LIN {X 0,Y 180.514,Z 1092.741,A -85,B 0,C 180,E1 5202.314,E2 5202.314} C_VEL
LIN {X 0,Y 161.576,Z 1104.142,A -85,B 0,C 180,E1 5198.165,E2 5198.165} C_VEL
LIN {X 0,Y 144.452,Z 1113.156,A -85,B 0,C 180,E1 5193.245,E2 5193.245} C_VEL
LIN {X 0,Y 126.484,Z 1121.616,A -85,B 0,C 180,E1 5186.105,E2 5186.105} C_VEL
LIN {X 0,Y 112.708,Z 1127.399,A -85,B 0,C 180,E1 5178.177,E2 5178.177} C_VEL
LIN {X 0,Y 100.075,Z 1132.394,A -85,B 0,C 180,E1 5166.833,E2 5166.833} C_VEL
LIN {X 0,Y 92.274,Z 1135.383,A -85,B 0,C 180,E1 5154.316,E2 5154.316} C_VEL
LIN {X 0,Y 88.588,Z 1137.104,A -85,B 0,C 180,E1 5140.404,E2 5140.404} C_VEL
LIN {X 0,Y 88.071,Z 1137.45,A -85,B 0,C 180,E1 5129.349,E2 5129.349} C_VEL
LIN {X 0,Y 88.847,Z 1136.939,A -85,B 0,C 180,E1 5117.653,E2 5117.653} C_VEL
LIN {X 0,Y 92.778,Z 1135.217,A -85,B 0,C 180,E1 5104.463,E2 5104.463} C_VEL
LIN {X 0,Y 101.858,Z 1131.792,A -85,B 0,C 180,E1 5091.078,E2 5091.078} C_VEL
LIN {X 0,Y 114.473,Z 1126.766,A -85,B 0,C 180,E1 5080.542,E2 5080.542} C_VEL
LIN {X 0,Y 130.71,Z 1119.847,A -85,B 0,C 180,E1 5071.884,E2 5071.884} C_VEL
LIN {X 0,Y 146.756,Z 1112.133,A -85,B 0,C 180,E1 5065.926,E2 5065.926} C_VEL
LIN {X 0,Y 165.729,Z 1101.922,A -85,B 0,C 180,E1 5060.745,E2 5060.745} C_VEL
LIN {X 0,Y 183.093,Z 1091.275,A -85,B 0,C 180,E1 5057.119,E2 5057.119} C_VEL
LIN {X 0,Y 202.882,Z 1077.554,A -85,B 0,C 180,E1 5053.854,E2 5053.854} C_VEL
LIN {X 0,Y 219.478,Z 1064.484,A -85,B 0,C 180,E1 5051.623,E2 5051.623} C_VEL
LIN {X 0,Y 238.252,Z 1047.708,A -85,B 0,C 180,E1 5049.514,E2 5049.514} C_VEL
LIN {X 0,Y 253.475,Z 1032.291,A -85,B 0,C 180,E1 5048.055,E2 5048.055} C_VEL
LIN {X 0,Y 269.807,Z 1013.44,A -85,B 0,C 180,E1 5046.686,E2 5046.686} C_VEL
LIN {X 0,Y 282.88,Z 996.295,A -85,B 0,C 180,E1 5045.721,E2 5045.721} C_VEL
LIN {X 0,Y 296.514,Z 975.768,A -85,B 0,C 180,E1 5044.812,E2 5044.812} C_VEL
LIN {X 0,Y 307.276,Z 957.078,A -85,B 0,C 180,E1 5044.155,E2 5044.155} C_VEL
LIN {X 0,Y 318.569,Z 934.064,A -85,B 0,C 180,E1 5043.522,E2 5043.522} C_VEL
LIN {X 0,Y 326.941,Z 913.681,A -85,B 0,C 180,E1 5043.088,E2 5043.088} C_VEL
LIN {X 0,Y 335.084,Z 889.205,A -85,B 0,C 180,E1 5042.688,E2 5042.688} C_VEL
LIN {X 0,Y 340.736,Z 867.45,A -85,B 0,C 180,E1 5042.416,E2 5042.416} C_VEL
LIN {X 0,Y 345.393,Z 842.416,A -85,B 0,C 180,E1 5042.144,E2 5042.144} C_VEL
LIN {X 0,Y 352.177,Z 788.71,A -85,B 0,C 180,E1 5041.569,E2 5041.569} C_VEL
LIN {X 0,Y 344.618,Z 847.74,A -85,B 0,C 180,E1 5040.925,E2 5040.925} C_VEL
LIN {X 0,Y 339.705,Z 871.733,A -85,B 0,C 180,E1 5040.649,E2 5040.649} C_VEL
LIN {X 0,Y 333.471,Z 894.758,A -85,B 0,C 180,E1 5040.334,E2 5040.334} C_VEL
LIN {X 0,Y 325.466,Z 917.45,A -85,B 0,C 180,E1 5039.929,E2 5039.929} C_VEL
LIN {X 0,Y 315.983,Z 939.81,A -85,B 0,C 180,E1 5039.422,E2 5039.422} C_VEL
LIN {X 0,Y 305.532,Z 960.244,A -85,B 0,C 180,E1 5038.827,E2 5038.827} C_VEL
LIN {X 0,Y 293.092,Z 981.341,A -85,B 0,C 180,E1 5038.045,E2 5038.045} C_VEL
LIN {X 0,Y 279.658,Z 1000.791,A -85,B 0,C 180,E1 5037.131,E2 5037.131} C_VEL
LIN {X 0,Y 264.625,Z 1019.965,A -85,B 0,C 180,E1 5035.975,E2 5035.975} C_VEL
LIN {X 0,Y 249.554,Z 1036.734,A -85,B 0,C 180,E1 5034.669,E2 5034.669} C_VEL
LIN {X 0,Y 232.717,Z 1053.447,A -85,B 0,C 180,E1 5032.987,E2 5032.987} C_VEL
LIN {X 0,Y 215.64,Z 1068.312,A -85,B 0,C 180,E1 5030.988,E2 5030.988} C_VEL
LIN {X 0,Y 210.299,Z 1072.727,A -85,B 0,C 180,E1 5030.284,E2 5030.284} C_VEL
LIN {X 0,Y 204.27,Z 1077.246,A -85,B 0,C 180,E1 5029.757,E2 5029.757} C_VEL
LIN {X 0,Y 187.534,Z 1088.286,A -85,B 0,C 180,E1 5029.208,E2 5029.208} C_VEL
LIN {X 0,Y 181.234,Z 1092.239,A -85,B 0,C 180,E1 5028.527,E2 5028.527} C_VEL
LIN {X 0,Y 163.079,Z 1103.329,A -85,B 0,C 180,E1 5025.077,E2 5025.077} C_VEL
LIN {X 0,Y 142.378,Z 1114.455,A -85,B 0,C 180,E1 5019.872,E2 5019.872} C_VEL
LIN {X 0,Y 125.566,Z 1122.468,A -85,B 0,C 180,E1 5014.025,E2 5014.025} C_VEL
LIN {X 0,Y 108.268,Z 1129.827,A -85,B 0,C 180,E1 5005.28,E2 5005.28} C_VEL
LIN {X 0,Y 95.103,Z 1135.026,A -85,B 0,C 180,E1 4994.783,E2 4994.783} C_VEL
LIN {X 0,Y 84.698,Z 1139.105,A -85,B 0,C 180,E1 4979.724,E2 4979.724} C_VEL
LIN {X 0,Y 80.754,Z 1140.969,A -85,B 0,C 180,E1 4966.546,E2 4966.546} C_VEL
LIN {X 0,Y 79.997,Z 1141.711,A -85,B 0,C 180,E1 4955.019,E2 4955.019} C_VEL
LIN {X 0,Y 80.026,Z 1141.802,A -85,B 0,C 180,E1 4947.852,E2 4947.852} C_VEL
LIN {X 0,Y 80.375,Z 1141.239,A -85,B 0,C 180,E1 4936.328,E2 4936.328} C_VEL
LIN {X 0,Y 83.833,Z 1139.429,A -85,B 0,C 180,E1 4922.279,E2 4922.279} C_VEL
LIN {X 0,Y 92.595,Z 1135.983,A -85,B 0,C 180,E1 4907.97,E2 4907.97} C_VEL
LIN {X 0,Y 105.649,Z 1130.794,A -85,B 0,C 180,E1 4896.441,E2 4896.441} C_VEL
LIN {X 0,Y 121.066,Z 1124.38,A -85,B 0,C 180,E1 4887.905,E2 4887.905} C_VEL
LIN {X 0,Y 139.45,Z 1115.772,A -85,B 0,C 180,E1 4881.009,E2 4881.009} C_VEL
LIN {X 0,Y 158.123,Z 1106.034,A -85,B 0,C 180,E1 4876.018,E2 4876.018} C_VEL
LIN {X 0,Y 176.98,Z 1094.75,A -85,B 0,C 180,E1 4872.201,E2 4872.201} C_VEL
LIN {X 0,Y 195.527,Z 1082.343,A -85,B 0,C 180,E1 4869.258,E2 4869.258} C_VEL
LIN {X 0,Y 214.497,Z 1067.805,A -85,B 0,C 180,E1 4866.823,E2 4866.823} C_VEL
LIN {X 0,Y 232.288,Z 1052.516,A -85,B 0,C 180,E1 4864.939,E2 4864.939} C_VEL
LIN {X 0,Y 249.412,Z 1035.598,A -85,B 0,C 180,E1 4863.395,E2 4863.395} C_VEL
LIN {X 0,Y 265.655,Z 1017.529,A -85,B 0,C 180,E1 4862.13,E2 4862.13} C_VEL
LIN {X 0,Y 280.026,Z 999.098,A -85,B 0,C 180,E1 4861.142,E2 4861.142} C_VEL
LIN {X 0,Y 293.973,Z 978.764,A -85,B 0,C 180,E1 4860.288,E2 4860.288} C_VEL
LIN {X 0,Y 305.646,Z 958.886,A -85,B 0,C 180,E1 4859.625,E2 4859.625} C_VEL
LIN {X 0,Y 316.509,Z 937.477,A -85,B 0,C 180,E1 4859.065,E2 4859.065} C_VEL
LIN {X 0,Y 325.559,Z 915.956,A -85,B 0,C 180,E1 4858.631,E2 4858.631} C_VEL
LIN {X 0,Y 330.238,Z 903.054,A -85,B 0,C 180,E1 4858.407,E2 4858.407} C_VEL
LIN {X 0,Y 321.662,Z 925.806,A -85,B 0,C 180,E1 4858.004,E2 4858.004} C_VEL
LIN {X 0,Y 311.963,Z 946.817,A -85,B 0,C 180,E1 4857.526,E2 4857.526} C_VEL
LIN {X 0,Y 300.406,Z 968.233,A -85,B 0,C 180,E1 4856.909,E2 4856.909} C_VEL
LIN {X 0,Y 288.154,Z 987.533,A -85,B 0,C 180,E1 4856.2,E2 4856.2} C_VEL
LIN {X 0,Y 273.899,Z 1007.211,A -85,B 0,C 180,E1 4855.283,E2 4855.283} C_VEL
LIN {X 0,Y 259.287,Z 1024.684,A -85,B 0,C 180,E1 4854.229,E2 4854.229} C_VEL
LIN {X 0,Y 242.854,Z 1042.089,A -85,B 0,C 180,E1 4852.868,E2 4852.868} C_VEL
LIN {X 0,Y 226.575,Z 1057.152,A -85,B 0,C 180,E1 4851.314,E2 4851.314} C_VEL
LIN {X 0,Y 208.615,Z 1071.963,A -85,B 0,C 180,E1 4849.286,E2 4849.286} C_VEL
LIN {X 0,Y 190.964,Z 1084.666,A -85,B 0,C 180,E1 4846.882,E2 4846.882} C_VEL
LIN {X 0,Y 171.93,Z 1096.865,A -85,B 0,C 180,E1 4843.657,E2 4843.657} C_VEL
LIN {X 0,Y 153.55,Z 1107.072,A -85,B 0,C 180,E1 4839.67,E2 4839.67} C_VEL
LIN {X 0,Y 134.485,Z 1116.453,A -85,B 0,C 180,E1 4834.11,E2 4834.11} C_VEL
LIN {X 0,Y 117.722,Z 1123.611,A -85,B 0,C 180,E1 4827.233,E2 4827.233} C_VEL
LIN {X 0,Y 101.608,Z 1129.793,A -85,B 0,C 180,E1 4817.233,E2 4817.233} C_VEL
LIN {X 0,Y 90.459,Z 1133.686,A -85,B 0,C 180,E1 4805.862,E2 4805.862} C_VEL
LIN {X 0,Y 82.662,Z 1136.478,A -85,B 0,C 180,E1 4790.536,E2 4790.536} C_VEL
LIN {X 0,Y 80.264,Z 1137.458,A -85,B 0,C 180,E1 4777.156,E2 4777.156} C_VEL
LIN {X 0,Y 80.087,Z 1137.594,A -85,B 0,C 180,E1 4767.137,E2 4767.137} C_VEL
LIN {X 0,Y 81.399,Z 1136.957,A -85,B 0,C 180,E1 4754.321,E2 4754.321} C_VEL
LIN {X 0,Y 86.185,Z 1135.212,A -85,B 0,C 180,E1 4740.839,E2 4740.839} C_VEL
LIN {X 0,Y 97.246,Z 1131.404,A -85,B 0,C 180,E1 4726.457,E2 4726.457} C_VEL
LIN {X 0,Y 110.682,Z 1126.484,A -85,B 0,C 180,E1 4716.484,E2 4716.484} C_VEL
LIN {X 0,Y 128.899,Z 1119.024,A -85,B 0,C 180,E1 4707.832,E2 4707.832} C_VEL
LIN {X 0,Y 145.872,Z 1111.156,A -85,B 0,C 180,E1 4702.275,E2 4702.275} C_VEL
LIN {X 0,Y 165.655,Z 1100.621,A -85,B 0,C 180,E1 4697.505,E2 4697.505} C_VEL
LIN {X 0,Y 183.74,Z 1089.709,A -85,B 0,C 180,E1 4694.175,E2 4694.175} C_VEL
LIN {X 0,Y 202.953,Z 1076.4,A -85,B 0,C 180,E1 4691.357,E2 4691.357} C_VEL
LIN {X 0,Y 220.831,Z 1062.434,A -85,B 0,C 180,E1 4689.221,E2 4689.221} C_VEL
LIN {X 0,Y 238.175,Z 1046.883,A -85,B 0,C 180,E1 4687.478,E2 4687.478} C_VEL
LIN {X 0,Y 254.406,Z 1030.543,A -85,B 0,C 180,E1 4686.084,E2 4686.084} C_VEL
LIN {X 0,Y 269.963,Z 1012.521,A -85,B 0,C 180,E1 4684.912,E2 4684.912} C_VEL
LIN {X 0,Y 284.154,Z 993.949,A -85,B 0,C 180,E1 4683.976,E2 4683.976} C_VEL
LIN {X 0,Y 297.427,Z 973.701,A -85,B 0,C 180,E1 4683.18,E2 4683.18} C_VEL
LIN {X 0,Y 309.271,Z 952.974,A -85,B 0,C 180,E1 4682.537,E2 4682.537} C_VEL
LIN {X 0,Y 319.664,Z 931.164,A -85,B 0,C 180,E1 4682.012,E2 4682.012} C_VEL
LIN {X 0,Y 328.842,Z 908.282,A -85,B 0,C 180,E1 4681.586,E2 4681.586} C_VEL
LIN {X 0,Y 329.621,Z 905.974,A -85,B 0,C 180,E1 4681.548,E2 4681.548} C_VEL
LIN {X 0,Y 320.528,Z 929.195,A -85,B 0,C 180,E1 4681.122,E2 4681.122} C_VEL
LIN {X 0,Y 311.488,Z 948.495,A -85,B 0,C 180,E1 4680.664,E2 4680.664} C_VEL
LIN {X 0,Y 298.969,Z 971.183,A -85,B 0,C 180,E1 4679.988,E2 4679.988} C_VEL
LIN {X 0,Y 286.993,Z 989.827,A -85,B 0,C 180,E1 4679.284,E2 4679.284} C_VEL
LIN {X 0,Y 271.594,Z 1010.601,A -85,B 0,C 180,E1 4678.286,E2 4678.286} C_VEL
LIN {X 0,Y 256.782,Z 1028.09,A -85,B 0,C 180,E1 4677.189,E2 4677.189} C_VEL
LIN {X 0,Y 239.636,Z 1045.793,A -85,B 0,C 180,E1 4675.745,E2 4675.745} C_VEL
LIN {X 0,Y 222.674,Z 1061.316,A -85,B 0,C 180,E1 4674.072,E2 4674.072} C_VEL
LIN {X 0,Y 204.021,Z 1076.268,A -85,B 0,C 180,E1 4671.887,E2 4671.887} C_VEL
LIN {X 0,Y 185.27,Z 1089.642,A -85,B 0,C 180,E1 4669.187,E2 4669.187} C_VEL
LIN {X 0,Y 181.234,Z 1092.239,A -85,B 0,C 180,E1 4668.527,E2 4668.527} C_VEL
LIN {X 0,Y 174.874,Z 1096.127,A -85,B 0,C 180,E1 4667.781,E2 4667.781} C_VEL
LIN {X 0,Y 156.317,Z 1105.93,A -85,B 0,C 180,E1 4666.648,E2 4666.648} C_VEL
LIN {X 0,Y 150.773,Z 1108.689,A -85,B 0,C 180,E1 4665.773,E2 4665.773} C_VEL
LIN {X 0,Y 131.4,Z 1118.23,A -85,B 0,C 180,E1 4660.663,E2 4660.663} C_VEL
LIN {X 0,Y 112.711,Z 1126.128,A -85,B 0,C 180,E1 4653.637,E2 4653.637} C_VEL
LIN {X 0,Y 96.223,Z 1132.453,A -85,B 0,C 180,E1 4644.148,E2 4644.148} C_VEL
LIN {X 0,Y 83.081,Z 1136.987,A -85,B 0,C 180,E1 4631.447,E2 4631.447} C_VEL
LIN {X 0,Y 74.722,Z 1140.085,A -85,B 0,C 180,E1 4615.354,E2 4615.354} C_VEL
LIN {X 0,Y 72.037,Z 1141.397,A -85,B 0,C 180,E1 4598.783,E2 4598.783} C_VEL
LIN {X 0,Y 72.05,Z 1141.64,A -85,B 0,C 180,E1 4589.205,E2 4589.205} C_VEL
LIN {X 0,Y 72.206,Z 1141.284,A -85,B 0,C 180,E1 4578.011,E2 4578.011} C_VEL
LIN {X 0,Y 76.063,Z 1139.453,A -85,B 0,C 180,E1 4560.896,E2 4560.896} C_VEL
LIN {X 0,Y 84.556,Z 1136.434,A -85,B 0,C 180,E1 4546.696,E2 4546.696} C_VEL
LIN {X 0,Y 99.622,Z 1131.08,A -85,B 0,C 180,E1 4533.506,E2 4533.506} C_VEL
LIN {X 0,Y 115.63,Z 1124.862,A -85,B 0,C 180,E1 4525.07,E2 4525.07} C_VEL
LIN {X 0,Y 135.793,Z 1115.982,A -85,B 0,C 180,E1 4518.015,E2 4518.015} C_VEL
LIN {X 0,Y 154.225,Z 1106.745,A -85,B 0,C 180,E1 4513.467,E2 4513.467} C_VEL
LIN {X 0,Y 174.479,Z 1095.102,A -85,B 0,C 180,E1 4509.705,E2 4509.705} C_VEL
LIN {X 0,Y 192.455,Z 1083.398,A -85,B 0,C 180,E1 4507.097,E2 4507.097} C_VEL
LIN {X 0,Y 211.73,Z 1069.117,A -85,B 0,C 180,E1 4504.83,E2 4504.83} C_VEL
LIN {X 0,Y 229.316,Z 1054.363,A -85,B 0,C 180,E1 4503.122,E2 4503.122} C_VEL
LIN {X 0,Y 247.593,Z 1036.838,A -85,B 0,C 180,E1 4501.62,E2 4501.62} C_VEL
LIN {X 0,Y 262.984,Z 1020.126,A -85,B 0,C 180,E1 4500.529,E2 4500.529} C_VEL
LIN {X 0,Y 278.479,Z 1000.799,A -85,B 0,C 180,E1 4499.559,E2 4499.559} C_VEL
LIN {X 0,Y 291.731,Z 981.983,A -85,B 0,C 180,E1 4498.822,E2 4498.822} C_VEL
LIN {X 0,Y 299.524,Z 969.498,A -85,B 0,C 180,E1 4498.416,E2 4498.416} C_VEL
LIN {X 0,Y 287.188,Z 988.671,A -85,B 0,C 180,E1 4497.766,E2 4497.766} C_VEL
LIN {X 0,Y 271.876,Z 1009.318,A -85,B 0,C 180,E1 4496.875,E2 4496.875} C_VEL
LIN {X 0,Y 257.62,Z 1026.066,A -85,B 0,C 180,E1 4495.939,E2 4495.939} C_VEL
LIN {X 0,Y 240.036,Z 1044.183,A -85,B 0,C 180,E1 4494.612,E2 4494.612} C_VEL
LIN {X 0,Y 223.564,Z 1059.076,A -85,B 0,C 180,E1 4493.168,E2 4493.168} C_VEL
LIN {X 0,Y 204.401,Z 1074.28,A -85,B 0,C 180,E1 4491.17,E2 4491.17} C_VEL
LIN {X 0,Y 186.475,Z 1086.779,A -85,B 0,C 180,E1 4488.891,E2 4488.891} C_VEL
LIN {X 0,Y 166.165,Z 1099.122,A -85,B 0,C 180,E1 4485.654,E2 4485.654} C_VEL
LIN {X 0,Y 147.885,Z 1108.844,A -85,B 0,C 180,E1 4481.879,E2 4481.879} C_VEL
LIN {X 0,Y 127.81,Z 1118.057,A -85,B 0,C 180,E1 4476.252,E2 4476.252} C_VEL
LIN {X 0,Y 110.494,Z 1125.014,A -85,B 0,C 180,E1 4469.281,E2 4469.281} C_VEL
LIN {X 0,Y 93.986,Z 1130.73,A -85,B 0,C 180,E1 4459.056,E2 4459.056} C_VEL
LIN {X 0,Y 81.705,Z 1134.671,A -85,B 0,C 180,E1 4445.974,E2 4445.974} C_VEL
LIN {X 0,Y 74.127,Z 1136.983,A -85,B 0,C 180,E1 4429.226,E2 4429.226} C_VEL
LIN {X 0,Y 72.169,Z 1137.731,A -85,B 0,C 180,E1 4415.566,E2 4415.566} C_VEL
LIN {X 0,Y 72.11,Z 1137.783,A -85,B 0,C 180,E1 4406.024,E2 4406.024} C_VEL
LIN {X 0,Y 73.663,Z 1137.168,A -85,B 0,C 180,E1 4392.625,E2 4392.625} C_VEL
LIN {X 0,Y 79.198,Z 1135.424,A -85,B 0,C 180,E1 4377.977,E2 4377.977} C_VEL
LIN {X 0,Y 91.511,Z 1131.617,A -85,B 0,C 180,E1 4362.939,E2 4362.939} C_VEL
LIN {X 0,Y 105.313,Z 1126.945,A -85,B 0,C 180,E1 4353.33,E2 4353.33} C_VEL
LIN {X 0,Y 124.481,Z 1119.586,A -85,B 0,C 180,E1 4344.814,E2 4344.814} C_VEL
LIN {X 0,Y 142.11,Z 1111.77,A -85,B 0,C 180,E1 4339.467,E2 4339.467} C_VEL
LIN {X 0,Y 162.482,Z 1101.351,A -85,B 0,C 180,E1 4334.948,E2 4334.948} C_VEL
LIN {X 0,Y 180.834,Z 1090.59,A -85,B 0,C 180,E1 4331.848,E2 4331.848} C_VEL
LIN {X 0,Y 200.88,Z 1077.094,A -85,B 0,C 180,E1 4329.165,E2 4329.165} C_VEL
LIN {X 0,Y 217.753,Z 1064.194,A -85,B 0,C 180,E1 4327.322,E2 4327.322} C_VEL
LIN {X 0,Y 236.117,Z 1048.215,A -85,B 0,C 180,E1 4325.636,E2 4325.636} C_VEL
LIN {X 0,Y 251.719,Z 1032.814,A -85,B 0,C 180,E1 4324.411,E2 4324.411} C_VEL
LIN {X 0,Y 268.408,Z 1014.018,A -85,B 0,C 180,E1 4323.267,E2 4323.267} C_VEL
LIN {X 0,Y 281.731,Z 996.907,A -85,B 0,C 180,E1 4322.465,E2 4322.465} C_VEL
LIN {X 0,Y 296.097,Z 975.666,A -85,B 0,C 180,E1 4321.686,E2 4321.686} C_VEL
LIN {X 0,Y 298.821,Z 971.242,A -85,B 0,C 180,E1 4321.534,E2 4321.534} C_VEL
LIN {X 0,Y 286.504,Z 990.236,A -85,B 0,C 180,E1 4320.884,E2 4320.884} C_VEL
LIN {X 0,Y 271.292,Z 1010.529,A -85,B 0,C 180,E1 4320,E2 4320} C_VEL
LIN {X 0,Y 256.462,Z 1027.865,A -85,B 0,C 180,E1 4319.015,E2 4319.015} C_VEL
LIN {X 0,Y 239.166,Z 1045.537,A -85,B 0,C 180,E1 4317.708,E2 4317.708} C_VEL
LIN {X 0,Y 222.457,Z 1060.645,A -85,B 0,C 180,E1 4316.234,E2 4316.234} C_VEL
LIN {X 0,Y 203.02,Z 1076.033,A -85,B 0,C 180,E1 4314.194,E2 4314.194} C_VEL
LIN {X 0,Y 183.897,Z 1089.41,A -85,B 0,C 180,E1 4311.721,E2 4311.721} C_VEL
LIN {X 0,Y 164.267,Z 1101.321,A -85,B 0,C 180,E1 4308.524,E2 4308.524} C_VEL
LIN {X 0,Y 150.773,Z 1108.689,A -85,B 0,C 180,E1 4305.773,E2 4305.773} C_VEL
LIN {X 0,Y 144.235,Z 1111.943,A -85,B 0,C 180,E1 4304.698,E2 4304.698} C_VEL
LIN {X 0,Y 126.056,Z 1119.34,A -85,B 0,C 180,E1 4302.811,E2 4302.811} C_VEL
LIN {X 0,Y 119.505,Z 1121.914,A -85,B 0,C 180,E1 4301.308,E2 4301.308} C_VEL
LIN {X 0,Y 99.764,Z 1129.392,A -85,B 0,C 180,E1 4293.127,E2 4293.127} C_VEL
LIN {X 0,Y 84.188,Z 1134.592,A -85,B 0,C 180,E1 4282.727,E2 4282.727} C_VEL
LIN {X 0,Y 70.92,Z 1138.676,A -85,B 0,C 180,E1 4266.31,E2 4266.31} C_VEL
LIN {X 0,Y 65.157,Z 1140.616,A -85,B 0,C 180,E1 4249.731,E2 4249.731} C_VEL
LIN {X 0,Y 64.002,Z 1141.34,A -85,B 0,C 180,E1 4234.48,E2 4234.48} C_VEL
LIN {X 0,Y 64.01,Z 1141.358,A -85,B 0,C 180,E1 4226.418,E2 4226.418} C_VEL
LIN {X 0,Y 64.853,Z 1140.74,A -85,B 0,C 180,E1 4212.04,E2 4212.04} C_VEL
LIN {X 0,Y 70.129,Z 1138.878,A -85,B 0,C 180,E1 4195.227,E2 4195.227} C_VEL
LIN {X 0,Y 81.732,Z 1135.362,A -85,B 0,C 180,E1 4179.506,E2 4179.506} C_VEL
LIN {X 0,Y 97.477,Z 1130.095,A -85,B 0,C 180,E1 4168.095,E2 4168.095} C_VEL
LIN {X 0,Y 115.923,Z 1123.31,A -85,B 0,C 180,E1 4159.918,E2 4159.918} C_VEL
LIN {X 0,Y 136.017,Z 1114.58,A -85,B 0,C 180,E1 4153.983,E2 4153.983} C_VEL
LIN {X 0,Y 156.238,Z 1104.587,A -85,B 0,C 180,E1 4149.744,E2 4149.744} C_VEL
LIN {X 0,Y 176.147,Z 1093.122,A -85,B 0,C 180,E1 4146.595,E2 4146.595} C_VEL
LIN {X 0,Y 196.539,Z 1079.763,A -85,B 0,C 180,E1 4144.084,E2 4144.084} C_VEL
LIN {X 0,Y 214.154,Z 1066.531,A -85,B 0,C 180,E1 4142.323,E2 4142.323} C_VEL
LIN {X 0,Y 233.22,Z 1050.344,A -85,B 0,C 180,E1 4140.737,E2 4140.737} C_VEL
LIN {X 0,Y 249.481,Z 1034.538,A -85,B 0,C 180,E1 4139.586,E2 4139.586} C_VEL
LIN {X 0,Y 266.559,Z 1015.697,A -85,B 0,C 180,E1 4138.535,E2 4138.535} C_VEL
LIN {X 0,Y 268.63,Z 1013.173,A -85,B 0,C 180,E1 4138.415,E2 4138.415} C_VEL
LIN {X 0,Y 252.23,Z 1031.685,A -85,B 0,C 180,E1 4137.415,E2 4137.415} C_VEL
LIN {X 0,Y 236.462,Z 1047.194,A -85,B 0,C 180,E1 4136.323,E2 4136.323} C_VEL
LIN {X 0,Y 217.869,Z 1063.371,A -85,B 0,C 180,E1 4134.816,E2 4134.816} C_VEL
LIN {X 0,Y 200.315,Z 1076.67,A -85,B 0,C 180,E1 4133.119,E2 4133.119} C_VEL
LIN {X 0,Y 180.289,Z 1090.048,A -85,B 0,C 180,E1 4130.745,E2 4130.745} C_VEL
LIN {X 0,Y 161.544,Z 1100.87,A -85,B 0,C 180,E1 4127.949,E2 4127.949} C_VEL
LIN {X 0,Y 140.545,Z 1111.428,A -85,B 0,C 180,E1 4123.832,E2 4123.832} C_VEL
LIN {X 0,Y 122.166,Z 1119.321,A -85,B 0,C 180,E1 4118.892,E2 4118.892} C_VEL
LIN {X 0,Y 101.879,Z 1126.809,A -85,B 0,C 180,E1 4110.867,E2 4110.867} C_VEL
LIN {X 0,Y 86.215,Z 1131.746,A -85,B 0,C 180,E1 4100.991,E2 4100.991} C_VEL
LIN {X 0,Y 72.486,Z 1135.588,A -85,B 0,C 180,E1 4085.406,E2 4085.406} C_VEL
LIN {X 0,Y 66.026,Z 1137.35,A -85,B 0,C 180,E1 4069.461,E2 4069.461} C_VEL
LIN {X 0,Y 64.127,Z 1137.983,A -85,B 0,C 180,E1 4054.471,E2 4054.471} C_VEL
LIN {X 0,Y 64.195,Z 1137.95,A -85,B 0,C 180,E1 4043.741,E2 4043.741} C_VEL
LIN {X 0,Y 66.437,Z 1137.251,A -85,B 0,C 180,E1 4028.826,E2 4028.826} C_VEL
LIN {X 0,Y 74.749,Z 1135.092,A -85,B 0,C 180,E1 4011.046,E2 4011.046} C_VEL
LIN {X 0,Y 88.134,Z 1131.229,A -85,B 0,C 180,E1 3997.424,E2 3997.424} C_VEL
LIN {X 0,Y 105.712,Z 1125.653,A -85,B 0,C 180,E1 3987.237,E2 3987.237} C_VEL
LIN {X 0,Y 124.692,Z 1118.416,A -85,B 0,C 180,E1 3980.246,E2 3980.246} C_VEL
LIN {X 0,Y 144.189,Z 1109.907,A -85,B 0,C 180,E1 3975.279,E2 3975.279} C_VEL
LIN {X 0,Y 163.554,Z 1099.943,A -85,B 0,C 180,E1 3971.639,E2 3971.639} C_VEL
LIN {X 0,Y 183.282,Z 1088.418,A -85,B 0,C 180,E1 3968.787,E2 3968.787} C_VEL
LIN {X 0,Y 202.316,Z 1075.48,A -85,B 0,C 180,E1 3966.591,E2 3966.591} C_VEL
LIN {X 0,Y 220.769,Z 1061.327,A -85,B 0,C 180,E1 3964.854,E2 3964.854} C_VEL
LIN {X 0,Y 238.409,Z 1045.714,A -85,B 0,C 180,E1 3963.456,E2 3963.456} C_VEL
LIN {X 0,Y 255.677,Z 1028.422,A -85,B 0,C 180,E1 3962.287,E2 3962.287} C_VEL
LIN {X 0,Y 268.069,Z 1014.309,A -85,B 0,C 180,E1 3961.539,E2 3961.539} C_VEL
LIN {X 0,Y 250.344,Z 1034.027,A -85,B 0,C 180,E1 3960.458,E2 3960.458} C_VEL
LIN {X 0,Y 233.993,Z 1049.955,A -85,B 0,C 180,E1 3959.31,E2 3959.31} C_VEL
LIN {X 0,Y 215.143,Z 1066.028,A -85,B 0,C 180,E1 3957.754,E2 3957.754} C_VEL
LIN {X 0,Y 197.459,Z 1079.343,A -85,B 0,C 180,E1 3956.006,E2 3956.006} C_VEL
LIN {X 0,Y 177.002,Z 1092.801,A -85,B 0,C 180,E1 3953.513,E2 3953.513} C_VEL
LIN {X 0,Y 157.715,Z 1103.936,A -85,B 0,C 180,E1 3950.512,E2 3950.512} C_VEL
LIN {X 0,Y 136.923,Z 1114.303,A -85,B 0,C 180,E1 3946.227,E2 3946.227} C_VEL
LIN {X 0,Y 119.505,Z 1121.914,A -85,B 0,C 180,E1 3941.308,E2 3941.308} C_VEL
LIN {X 0,Y 112.983,Z 1124.395,A -85,B 0,C 180,E1 3939.62,E2 3939.62} C_VEL
LIN {X 0,Y 93.756,Z 1130.131,A -85,B 0,C 180,E1 3935.716,E2 3935.716} C_VEL
LIN {X 0,Y 88.399,Z 1131.771,A -85,B 0,C 180,E1 3933.446,E2 3933.446} C_VEL
LIN {X 0,Y 71.565,Z 1136.555,A -85,B 0,C 180,E1 3920.215,E2 3920.215} C_VEL
LIN {X 0,Y 60.349,Z 1139.656,A -85,B 0,C 180,E1 3902.018,E2 3902.018} C_VEL
LIN {X 0,Y 56.141,Z 1140.974,A -85,B 0,C 180,E1 3881.298,E2 3881.298} C_VEL
LIN {X 0,Y 56.048,Z 1141.22,A -85,B 0,C 180,E1 3868.978,E2 3868.978} C_VEL
LIN {X 0,Y 56.464,Z 1140.859,A -85,B 0,C 180,E1 3854.596,E2 3854.596} C_VEL
LIN {X 0,Y 62.419,Z 1138.978,A -85,B 0,C 180,E1 3833.221,E2 3833.221} C_VEL
LIN {X 0,Y 74.066,Z 1135.834,A -85,B 0,C 180,E1 3817.203,E2 3817.203} C_VEL
LIN {X 0,Y 92.256,Z 1130.401,A -85,B 0,C 180,E1 3804.437,E2 3804.437} C_VEL
LIN {X 0,Y 110.863,Z 1123.983,A -85,B 0,C 180,E1 3796.775,E2 3796.775} C_VEL
LIN {X 0,Y 131.47,Z 1115.597,A -85,B 0,C 180,E1 3791.155,E2 3791.155} C_VEL
LIN {X 0,Y 151.224,Z 1106.295,A -85,B 0,C 180,E1 3787.341,E2 3787.341} C_VEL
LIN {X 0,Y 172.46,Z 1094.636,A -85,B 0,C 180,E1 3784.268,E2 3784.268} C_VEL
LIN {X 0,Y 192.105,Z 1082.284,A -85,B 0,C 180,E1 3782.069,E2 3782.069} C_VEL
LIN {X 0,Y 212.07,Z 1067.772,A -85,B 0,C 180,E1 3780.27,E2 3780.27} C_VEL
LIN {X 0,Y 231.021,Z 1052.144,A -85,B 0,C 180,E1 3778.868,E2 3778.868} C_VEL
LIN {X 0,Y 237.881,Z 1045.788,A -85,B 0,C 180,E1 3778.4,E2 3778.4} C_VEL
LIN {X 0,Y 220.246,Z 1061.249,A -85,B 0,C 180,E1 3777.171,E2 3777.171} C_VEL
LIN {X 0,Y 201.566,Z 1075.444,A -85,B 0,C 180,E1 3775.628,E2 3775.628} C_VEL
LIN {X 0,Y 182.098,Z 1088.498,A -85,B 0,C 180,E1 3773.652,E2 3773.652} C_VEL
LIN {X 0,Y 161.941,Z 1100.077,A -85,B 0,C 180,E1 3771.081,E2 3771.081} C_VEL
LIN {X 0,Y 141.269,Z 1110.442,A -85,B 0,C 180,E1 3767.623,E2 3767.623} C_VEL
LIN {X 0,Y 120.371,Z 1119.187,A -85,B 0,C 180,E1 3762.8,E2 3762.8} C_VEL
LIN {X 0,Y 100.623,Z 1126.278,A -85,B 0,C 180,E1 3756.093,E2 3756.093} C_VEL
LIN {X 0,Y 82.755,Z 1131.562,A -85,B 0,C 180,E1 3746.481,E2 3746.481} C_VEL
LIN {X 0,Y 67.582,Z 1135.475,A -85,B 0,C 180,E1 3731.743,E2 3731.743} C_VEL
LIN {X 0,Y 58.733,Z 1137.498,A -85,B 0,C 180,E1 3713.052,E2 3713.052} C_VEL
LIN {X 0,Y 56.186,Z 1138.172,A -85,B 0,C 180,E1 3696.13,E2 3696.13} C_VEL
LIN {X 0,Y 56.144,Z 1138.202,A -85,B 0,C 180,E1 3684.891,E2 3684.891} C_VEL
LIN {X 0,Y 58.455,Z 1137.59,A -85,B 0,C 180,E1 3667.894,E2 3667.894} C_VEL
LIN {X 0,Y 65.999,Z 1135.848,A -85,B 0,C 180,E1 3650.483,E2 3650.483} C_VEL
LIN {X 0,Y 81.993,Z 1131.844,A -85,B 0,C 180,E1 3633.978,E2 3633.978} C_VEL
LIN {X 0,Y 98.932,Z 1126.877,A -85,B 0,C 180,E1 3624.546,E2 3624.546} C_VEL
LIN {X 0,Y 119.44,Z 1119.672,A -85,B 0,C 180,E1 3617.378,E2 3617.378} C_VEL
LIN {X 0,Y 138.454,Z 1111.805,A -85,B 0,C 180,E1 3612.85,E2 3612.85} C_VEL
LIN {X 0,Y 160.007,Z 1101.287,A -85,B 0,C 180,E1 3609.122,E2 3609.122} C_VEL
LIN {X 0,Y 179.17,Z 1090.47,A -85,B 0,C 180,E1 3606.604,E2 3606.604} C_VEL
LIN {X 0,Y 199.588,Z 1077.1,A -85,B 0,C 180,E1 3604.476,E2 3604.476} C_VEL
LIN {X 0,Y 217.271,Z 1063.907,A -85,B 0,C 180,E1 3602.978,E2 3602.978} C_VEL
LIN {X 0,Y 236.072,Z 1047.803,A -85,B 0,C 180,E1 3601.641,E2 3601.641} C_VEL
LIN {X 0,Y 237.474,Z 1046.507,A -85,B 0,C 180,E1 3601.545,E2 3601.545} C_VEL
LIN {X 0,Y 218.979,Z 1062.668,A -85,B 0,C 180,E1 3600.254,E2 3600.254} C_VEL
LIN {X 0,Y 200.032,Z 1076.979,A -85,B 0,C 180,E1 3598.679,E2 3598.679} C_VEL
LIN {X 0,Y 180.288,Z 1090.178,A -85,B 0,C 180,E1 3596.655,E2 3596.655} C_VEL
LIN {X 0,Y 159.857,Z 1101.919,A -85,B 0,C 180,E1 3594.008,E2 3594.008} C_VEL
LIN {X 0,Y 137.989,Z 1112.842,A -85,B 0,C 180,E1 3590.226,E2 3590.226} C_VEL
LIN {X 0,Y 118.709,Z 1121.049,A -85,B 0,C 180,E1 3585.617,E2 3585.617} C_VEL
LIN {X 0,Y 97.947,Z 1128.65,A -85,B 0,C 180,E1 3578.275,E2 3578.275} C_VEL
LIN {X 0,Y 88.399,Z 1131.771,A -85,B 0,C 180,E1 3573.446,E2 3573.446} C_VEL
LIN {X 0,Y 82.239,Z 1133.541,A -85,B 0,C 180,E1 3570.499,E2 3570.499} C_VEL
LIN {X 0,Y 64.165,Z 1137.152,A -85,B 0,C 180,E1 3562.11,E2 3562.11} C_VEL
LIN {X 0,Y 59.663,Z 1137.998,A -85,B 0,C 180,E1 3557.607,E2 3557.607} C_VEL
LIN {X 0,Y 50.41,Z 1140.116,A -85,B 0,C 180,E1 3537.143,E2 3537.143} C_VEL
LIN {X 0,Y 48.023,Z 1140.894,A -85,B 0,C 180,E1 3517.177,E2 3517.177} C_VEL
LIN {X 0,Y 48.026,Z 1140.986,A -85,B 0,C 180,E1 3507.614,E2 3507.614} C_VEL
LIN {X 0,Y 49.207,Z 1140.46,A -85,B 0,C 180,E1 3488.545,E2 3488.545} C_VEL
LIN {X 0,Y 56.888,Z 1138.568,A -85,B 0,C 180,E1 3466.726,E2 3466.726} C_VEL
LIN {X 0,Y 71.563,Z 1135.116,A -85,B 0,C 180,E1 3449.972,E2 3449.972} C_VEL
LIN {X 0,Y 90.001,Z 1129.92,A -85,B 0,C 180,E1 3439.208,E2 3439.208} C_VEL
LIN {X 0,Y 110.446,Z 1123.189,A -85,B 0,C 180,E1 3432.11,E2 3432.11} C_VEL
LIN {X 0,Y 132.029,Z 1114.547,A -85,B 0,C 180,E1 3427.205,E2 3427.205} C_VEL
LIN {X 0,Y 153.784,Z 1104.403,A -85,B 0,C 180,E1 3423.728,E2 3423.728} C_VEL
LIN {X 0,Y 174.027,Z 1093.24,A -85,B 0,C 180,E1 3421.304,E2 3421.304} C_VEL
LIN {X 0,Y 194.27,Z 1080.542,A -85,B 0,C 180,E1 3419.41,E2 3419.41} C_VEL
LIN {X 0,Y 207.061,Z 1071.488,A -85,B 0,C 180,E1 3418.382,E2 3418.382} C_VEL
LIN {X 0,Y 187.279,Z 1084.961,A -85,B 0,C 180,E1 3416.767,E2 3416.767} C_VEL
LIN {X 0,Y 166.709,Z 1097.251,A -85,B 0,C 180,E1 3414.65,E2 3414.65} C_VEL
LIN {X 0,Y 145.467,Z 1107.96,A -85,B 0,C 180,E1 3411.815,E2 3411.815} C_VEL
LIN {X 0,Y 123.762,Z 1117.322,A -85,B 0,C 180,E1 3407.846,E2 3407.846} C_VEL
LIN {X 0,Y 103.744,Z 1124.482,A -85,B 0,C 180,E1 3402.586,E2 3402.586} C_VEL
LIN {X 0,Y 82.505,Z 1130.772,A -85,B 0,C 180,E1 3393.743,E2 3393.743} C_VEL
LIN {X 0,Y 66.095,Z 1134.721,A -85,B 0,C 180,E1 3381.665,E2 3381.665} C_VEL
LIN {X 0,Y 52.795,Z 1137.454,A -85,B 0,C 180,E1 3360.754,E2 3360.754} C_VEL
LIN {X 0,Y 48.469,Z 1138.32,A -85,B 0,C 180,E1 3340.7,E2 3340.7} C_VEL
LIN {X 0,Y 48.114,Z 1138.446,A -85,B 0,C 180,E1 3325.964,E2 3325.964} C_VEL
LIN {X 0,Y 50.771,Z 1137.866,A -85,B 0,C 180,E1 3305.57,E2 3305.57} C_VEL
LIN {X 0,Y 59.392,Z 1136.169,A -85,B 0,C 180,E1 3286.35,E2 3286.35} C_VEL
LIN {X 0,Y 75.437,Z 1132.661,A -85,B 0,C 180,E1 3270.508,E2 3270.508} C_VEL
LIN {X 0,Y 93.251,Z 1127.834,A -85,B 0,C 180,E1 3261.114,E2 3261.114} C_VEL
LIN {X 0,Y 113.602,Z 1121.278,A -85,B 0,C 180,E1 3254.49,E2 3254.49} C_VEL
LIN {X 0,Y 134.032,Z 1113.218,A -85,B 0,C 180,E1 3250.023,E2 3250.023} C_VEL
LIN {X 0,Y 155.722,Z 1103.189,A -85,B 0,C 180,E1 3246.637,E2 3246.637} C_VEL
LIN {X 0,Y 175.477,Z 1092.395,A -85,B 0,C 180,E1 3244.305,E2 3244.305} C_VEL
LIN {X 0,Y 196.15,Z 1079.414,A -85,B 0,C 180,E1 3242.389,E2 3242.389} C_VEL
LIN {X 0,Y 206.745,Z 1071.997,A -85,B 0,C 180,E1 3241.552,E2 3241.552} C_VEL
LIN {X 0,Y 186.981,Z 1085.496,A -85,B 0,C 180,E1 3239.946,E2 3239.946} C_VEL
LIN {X 0,Y 166.104,Z 1098.031,A -85,B 0,C 180,E1 3237.807,E2 3237.807} C_VEL
LIN {X 0,Y 145.523,Z 1108.565,A -85,B 0,C 180,E1 3235.07,E2 3235.07} C_VEL
LIN {X 0,Y 123.484,Z 1118.299,A -85,B 0,C 180,E1 3231.069,E2 3231.069} C_VEL
LIN {X 0,Y 103.177,Z 1125.786,A -85,B 0,C 180,E1 3225.722,E2 3225.722} C_VEL
LIN {X 0,Y 81.666,Z 1132.447,A -85,B 0,C 180,E1 3216.676,E2 3216.676} C_VEL
LIN {X 0,Y 65.24,Z 1136.673,A -85,B 0,C 180,E1 3204.322,E2 3204.322} C_VEL
LIN {X 0,Y 59.663,Z 1137.998,A -85,B 0,C 180,E1 3197.607,E2 3197.607} C_VEL
LIN {X 0,Y 54.827,Z 1138.903,A -85,B 0,C 180,E1 3191.586,E2 3191.586} C_VEL
LIN {X 0,Y 45.915,Z 1140.005,A -85,B 0,C 180,E1 3180.15,E2 3180.15} C_VEL
LIN {X 0,Y 40.878,Z 1140.521,A -85,B 0,C 180,E1 3167.711,E2 3167.711} C_VEL
LIN {X 0,Y 40.162,Z 1140.616,A -85,B 0,C 180,E1 3162.265,E2 3162.265} C_VEL
LIN {X 0,Y 40.028,Z 1140.786,A -85,B 0,C 180,E1 3147.709,E2 3147.709} C_VEL
LIN {X 0,Y 41.745,Z 1140.246,A -85,B 0,C 180,E1 3124.459,E2 3124.459} C_VEL
LIN {X 0,Y 51.217,Z 1138.353,A -85,B 0,C 180,E1 3100.414,E2 3100.414} C_VEL
LIN {X 0,Y 67.817,Z 1134.9,A -85,B 0,C 180,E1 3083.917,E2 3083.917} C_VEL
LIN {X 0,Y 87.624,Z 1129.701,A -85,B 0,C 180,E1 3074.081,E2 3074.081} C_VEL
LIN {X 0,Y 109.007,Z 1122.97,A -85,B 0,C 180,E1 3067.839,E2 3067.839} C_VEL
LIN {X 0,Y 131.246,Z 1114.323,A -85,B 0,C 180,E1 3063.606,E2 3063.606} C_VEL
LIN {X 0,Y 152.995,Z 1104.421,A -85,B 0,C 180,E1 3060.69,E2 3060.69} C_VEL
LIN {X 0,Y 174.035,Z 1093.007,A -85,B 0,C 180,E1 3058.579,E2 3058.579} C_VEL
LIN {X 0,Y 176.215,Z 1091.748,A -85,B 0,C 180,E1 3058.374,E2 3058.374} C_VEL
LIN {X 0,Y 156.288,Z 1102.557,A -85,B 0,C 180,E1 3056.424,E2 3056.424} C_VEL
LIN {X 0,Y 133.842,Z 1112.882,A -85,B 0,C 180,E1 3053.517,E2 3053.517} C_VEL
LIN {X 0,Y 113.55,Z 1120.737,A -85,B 0,C 180,E1 3049.856,E2 3049.856} C_VEL
LIN {X 0,Y 91.562,Z 1127.703,A -85,B 0,C 180,E1 3043.944,E2 3043.944} C_VEL
LIN {X 0,Y 72.499,Z 1132.594,A -85,B 0,C 180,E1 3035.542,E2 3035.542} C_VEL
LIN {X 0,Y 53.844,Z 1136.336,A -85,B 0,C 180,E1 3019.586,E2 3019.586} C_VEL
LIN {X 0,Y 43.223,Z 1138.115,A -85,B 0,C 180,E1 2997.559,E2 2997.559} C_VEL
LIN {X 0,Y 40.097,Z 1138.677,A -85,B 0,C 180,E1 2972.859,E2 2972.859} C_VEL
LIN {X 0,Y 41.088,Z 1138.479,A -85,B 0,C 180,E1 2953.021,E2 2953.021} C_VEL
LIN {X 0,Y 50.149,Z 1137.035,A -85,B 0,C 180,E1 2925.745,E2 2925.745} C_VEL
LIN {X 0,Y 65.254,Z 1134.203,A -85,B 0,C 180,E1 2909.141,E2 2909.141} C_VEL
LIN {X 0,Y 86.174,Z 1129.292,A -85,B 0,C 180,E1 2897.925,E2 2897.925} C_VEL
LIN {X 0,Y 105.28,Z 1123.628,A -85,B 0,C 180,E1 2891.974,E2 2891.974} C_VEL
LIN {X 0,Y 128.033,Z 1115.43,A -85,B 0,C 180,E1 2887.329,E2 2887.329} C_VEL
LIN {X 0,Y 148.424,Z 1106.544,A -85,B 0,C 180,E1 2884.408,E2 2884.408} C_VEL
LIN {X 0,Y 171.087,Z 1094.886,A -85,B 0,C 180,E1 2882.003,E2 2882.003} C_VEL
LIN {X 0,Y 175.723,Z 1092.239,A -85,B 0,C 180,E1 2881.557,E2 2881.557} C_VEL
LIN {X 0,Y 155.942,Z 1103.059,A -85,B 0,C 180,E1 2879.633,E2 2879.633} C_VEL
LIN {X 0,Y 133.208,Z 1113.642,A -85,B 0,C 180,E1 2876.69,E2 2876.69} C_VEL
LIN {X 0,Y 111.973,Z 1122.013,A -85,B 0,C 180,E1 2872.818,E2 2872.818} C_VEL
LIN {X 0,Y 90.346,Z 1129.003,A -85,B 0,C 180,E1 2866.888,E2 2866.888} C_VEL
LIN {X 0,Y 70.269,Z 1134.37,A -85,B 0,C 180,E1 2857.656,E2 2857.656} C_VEL
LIN {X 0,Y 52.46,Z 1138.152,A -85,B 0,C 180,E1 2841.394,E2 2841.394} C_VEL
LIN {X 0,Y 42.63,Z 1140.05,A -85,B 0,C 180,E1 2819.509,E2 2819.509} C_VEL
LIN {X 0,Y 40.162,Z 1140.616,A -85,B 0,C 180,E1 2802.265,E2 2802.265} C_VEL
LIN {X 0,Y 39.157,Z 1140.765,A -85,B 0,C 180,E1 2793.647,E2 2793.647} C_VEL
LIN {X 0,Y 37.136,Z 1140.649,A -85,B 0,C 180,E1 2782.313,E2 2782.313} C_VEL
LIN {X 0,Y 36.1,Z 1139.835,A -85,B 0,C 180,E1 2754.261,E2 2754.261} C_VEL
LIN {X 0,Y 37.879,Z 1139.482,A -85,B 0,C 180,E1 2747.705,E2 2747.705} C_VEL
LIN {X 0,Y 53.938,Z 1136.85,A -85,B 0,C 180,E1 2724.72,E2 2724.72} C_VEL
LIN {X 0,Y 73.876,Z 1132.584,A -85,B 0,C 180,E1 2712.966,E2 2712.966} C_VEL
LIN {X 0,Y 96.506,Z 1126.481,A -85,B 0,C 180,E1 2705.926,E2 2705.926} C_VEL
LIN {X 0,Y 118.046,Z 1119.176,A -85,B 0,C 180,E1 2701.793,E2 2701.793} C_VEL
LIN {X 0,Y 142.022,Z 1109.352,A -85,B 0,C 180,E1 2698.696,E2 2698.696} C_VEL
LIN {X 0,Y 145.044,Z 1107.951,A -85,B 0,C 180,E1 2698.358,E2 2698.358} C_VEL
LIN {X 0,Y 123.336,Z 1117.062,A -85,B 0,C 180,E1 2695.689,E2 2695.689} C_VEL
LIN {X 0,Y 101.034,Z 1124.617,A -85,B 0,C 180,E1 2691.755,E2 2691.755} C_VEL
LIN {X 0,Y 78.519,Z 1130.799,A -85,B 0,C 180,E1 2685.425,E2 2685.425} C_VEL
LIN {X 0,Y 59.21,Z 1134.818,A -85,B 0,C 180,E1 2675.771,E2 2675.771} C_VEL
LIN {X 0,Y 41.517,Z 1137.687,A -85,B 0,C 180,E1 2656.263,E2 2656.263} C_VEL
LIN {X 0,Y 33.023,Z 1138.721,A -85,B 0,C 180,E1 2627.625,E2 2627.625} C_VEL
LIN {X 0,Y 32.105,Z 1138.896,A -85,B 0,C 180,E1 2606.429,E2 2606.429} C_VEL
LIN {X 0,Y 36.236,Z 1138.353,A -85,B 0,C 180,E1 2576.504,E2 2576.504} C_VEL
LIN {X 0,Y 48.94,Z 1136.594,A -85,B 0,C 180,E1 2553.105,E2 2553.105} C_VEL
LIN {X 0,Y 68.611,Z 1133.09,A -85,B 0,C 180,E1 2538.689,E2 2538.689} C_VEL
LIN {X 0,Y 88.686,Z 1128.264,A -85,B 0,C 180,E1 2531.221,E2 2531.221} C_VEL
LIN {X 0,Y 111.024,Z 1121.578,A -85,B 0,C 180,E1 2526.204,E2 2526.204} C_VEL
LIN {X 0,Y 132.172,Z 1113.654,A -85,B 0,C 180,E1 2523.034,E2 2523.034} C_VEL
LIN {X 0,Y 144.739,Z 1108.258,A -85,B 0,C 180,E1 2521.583,E2 2521.583} C_VEL
LIN {X 0,Y 122.014,Z 1117.861,A -85,B 0,C 180,E1 2518.795,E2 2518.795} C_VEL
LIN {X 0,Y 100.38,Z 1125.348,A -85,B 0,C 180,E1 2514.944,E2 2514.944} C_VEL
LIN {X 0,Y 77.556,Z 1131.8,A -85,B 0,C 180,E1 2508.475,E2 2508.475} C_VEL
LIN {X 0,Y 58.042,Z 1136.075,A -85,B 0,C 180,E1 2498.476,E2 2498.476} C_VEL
LIN {X 0,Y 40.39,Z 1139.172,A -85,B 0,C 180,E1 2477.961,E2 2477.961} C_VEL
LIN {X 0,Y 32.46,Z 1140.375,A -85,B 0,C 180,E1 2447.271,E2 2447.271} C_VEL
LIN {X 0,Y 32.035,Z 1140.59,A -85,B 0,C 180,E1 2428.211,E2 2428.211} C_VEL
LIN {X 0,Y 34.233,Z 1140.105,A -85,B 0,C 180,E1 2400.228,E2 2400.228} C_VEL
LIN {X 0,Y 37.879,Z 1139.482,A -85,B 0,C 180,E1 2387.705,E2 2387.705} C_VEL
LIN {X 0,Y 41.456,Z 1138.856,A -85,B 0,C 180,E1 2377.779,E2 2377.779} C_VEL
LIN {X 0,Y 53.388,Z 1136.261,A -85,B 0,C 180,E1 2355.578,E2 2355.578} C_VEL
LIN {X 0,Y 58.399,Z 1135.283,A -85,B 0,C 180,E1 2352.09,E2 2352.09} C_VEL
LIN {X 0,Y 82.18,Z 1130.046,A -85,B 0,C 180,E1 2343.881,E2 2343.881} C_VEL
LIN {X 0,Y 103.991,Z 1123.774,A -85,B 0,C 180,E1 2339.667,E2 2339.667} C_VEL
LIN {X 0,Y 113.41,Z 1120.623,A -85,B 0,C 180,E1 2338.343,E2 2338.343} C_VEL
LIN {X 0,Y 88.422,Z 1128.141,A -85,B 0,C 180,E1 2334.159,E2 2334.159} C_VEL
LIN {X 0,Y 67.402,Z 1133.023,A -85,B 0,C 180,E1 2328.265,E2 2328.265} C_VEL
LIN {X 0,Y 45.042,Z 1136.762,A -85,B 0,C 180,E1 2315.527,E2 2315.527} C_VEL
LIN {X 0,Y 29.855,Z 1138.539,A -85,B 0,C 180,E1 2292.055,E2 2292.055} C_VEL
LIN {X 0,Y 24.123,Z 1139.097,A -85,B 0,C 180,E1 2254.755,E2 2254.755} C_VEL
LIN {X 0,Y 25.782,Z 1138.921,A -85,B 0,C 180,E1 2224.748,E2 2224.748} C_VEL
LIN {X 0,Y 39.376,Z 1137.569,A -85,B 0,C 180,E1 2190.301,E2 2190.301} C_VEL
LIN {X 0,Y 58.149,Z 1134.785,A -85,B 0,C 180,E1 2175.648,E2 2175.648} C_VEL
LIN {X 0,Y 80.695,Z 1130.219,A -85,B 0,C 180,E1 2167.57,E2 2167.57} C_VEL
LIN {X 0,Y 102.15,Z 1124.356,A -85,B 0,C 180,E1 2163.215,E2 2163.215} C_VEL
LIN {X 0,Y 113.032,Z 1120.889,A -85,B 0,C 180,E1 2161.598,E2 2161.598} C_VEL
LIN {X 0,Y 89.065,Z 1128.306,A -85,B 0,C 180,E1 2157.668,E2 2157.668} C_VEL
LIN {X 0,Y 67.683,Z 1133.508,A -85,B 0,C 180,E1 2151.815,E2 2151.815} C_VEL
LIN {X 0,Y 44.955,Z 1137.601,A -85,B 0,C 180,E1 2139.095,E2 2139.095} C_VEL
LIN {X 0,Y 30.123,Z 1139.549,A -85,B 0,C 180,E1 2116.908,E2 2116.908} C_VEL
LIN {X 0,Y 24.02,Z 1140.338,A -85,B 0,C 180,E1 2077.174,E2 2077.174} C_VEL
LIN {X 0,Y 24.02,Z 1140.33,A -85,B 0,C 180,E1 2062.826,E2 2062.826} C_VEL
LIN {X 0,Y 29.546,Z 1139.599,A -85,B 0,C 180,E1 2024.709,E2 2024.709} C_VEL
LIN {X 0,Y 44.954,Z 1137.56,A -85,B 0,C 180,E1 2000.903,E2 2000.903} C_VEL
LIN {X 0,Y 58.399,Z 1135.283,A -85,B 0,C 180,E1 1992.09,E2 1992.09} C_VEL
LIN {X 0,Y 62.551,Z 1134.488,A -85,B 0,C 180,E1 1989.182,E2 1989.182} C_VEL
LIN {X 0,Y 72.556,Z 1132.055,A -85,B 0,C 180,E1 1980.51,E2 1980.51} C_VEL
LIN {X 0,Y 76.552,Z 1131.174,A -85,B 0,C 180,E1 1979.079,E2 1979.079} C_VEL
LIN {X 0,Y 80.654,Z 1130.183,A -85,B 0,C 180,E1 1978.264,E2 1978.264} C_VEL
LIN {X 0,Y 57.474,Z 1134.782,A -85,B 0,C 180,E1 1972.59,E2 1972.59} C_VEL
LIN {X 0,Y 36.876,Z 1137.629,A -85,B 0,C 180,E1 1961.626,E2 1961.626} C_VEL
LIN {X 0,Y 19.339,Z 1139.103,A -85,B 0,C 180,E1 1928.347,E2 1928.347} C_VEL
LIN {X 0,Y 16.101,Z 1139.337,A -85,B 0,C 180,E1 1886.44,E2 1886.44} C_VEL
LIN {X 0,Y 23.02,Z 1138.906,A -85,B 0,C 180,E1 1838.569,E2 1838.569} C_VEL
LIN {X 0,Y 41.392,Z 1137.129,A -85,B 0,C 180,E1 1814.923,E2 1814.923} C_VEL
LIN {X 0,Y 64.263,Z 1133.719,A -85,B 0,C 180,E1 1805.252,E2 1805.252} C_VEL
LIN {X 0,Y 80.566,Z 1130.3,A -85,B 0,C 180,E1 1801.649,E2 1801.649} C_VEL
LIN {X 0,Y 57.135,Z 1135.142,A -85,B 0,C 180,E1 1795.98,E2 1795.98} C_VEL
LIN {X 0,Y 36.26,Z 1138.226,A -85,B 0,C 180,E1 1784.827,E2 1784.827} C_VEL
LIN {X 0,Y 18.72,Z 1139.886,A -85,B 0,C 180,E1 1749.862,E2 1749.862} C_VEL
LIN {X 0,Y 16.049,Z 1140.191,A -85,B 0,C 180,E1 1710,E2 1710} C_VEL
LIN {X 0,Y 21.662,Z 1139.677,A -85,B 0,C 180,E1 1658.308,E2 1658.308} C_VEL
LIN {X 0,Y 39.919,Z 1137.705,A -85,B 0,C 180,E1 1632.344,E2 1632.344} C_VEL
LIN {X 0,Y 62.051,Z 1134.248,A -85,B 0,C 180,E1 1622.475,E2 1622.475} C_VEL
LIN {X 0,Y 76.552,Z 1131.174,A -85,B 0,C 180,E1 1619.079,E2 1619.079} C_VEL
LIN {X 0,Y 75.427,Z 1131.413,A -85,B 0,C 180,E1 1618.428,E2 1618.428} C_VEL
LIN {X 0,Y 66.799,Z 1133.182,A -85,B 0,C 180,E1 1617.529,E2 1617.529} C_VEL
LIN {X 0,Y 44.151,Z 1136.84,A -85,B 0,C 180,E1 1616.617,E2 1616.617} C_VEL
LIN {X 0,Y 34.47,Z 1137.921,A -85,B 0,C 180,E1 1613.948,E2 1613.948} C_VEL
LIN {X 0,Y 13.164,Z 1139.334,A -85,B 0,C 180,E1 1586.671,E2 1586.671} C_VEL
LIN {X 0,Y 8.129,Z 1139.547,A -85,B 0,C 180,E1 1522.935,E2 1522.935} C_VEL
LIN {X 0,Y 19.96,Z 1139.053,A -85,B 0,C 180,E1 1457.865,E2 1457.865} C_VEL
LIN {X 0,Y 40.076,Z 1137.342,A -85,B 0,C 180,E1 1443.616,E2 1443.616} C_VEL
LIN {X 0,Y 45.798,Z 1136.715,A -85,B 0,C 180,E1 1441.722,E2 1441.722} C_VEL
LIN {X 0,Y 24.295,Z 1138.973,A -85,B 0,C 180,E1 1431.02,E2 1431.02} C_VEL
LIN {X 0,Y 9.432,Z 1139.836,A -85,B 0,C 180,E1 1389.498,E2 1389.498} C_VEL
LIN {X 0,Y 8.015,Z 1139.959,A -85,B 0,C 180,E1 1342.833,E2 1342.833} C_VEL
LIN {X 0,Y 20.532,Z 1139.243,A -85,B 0,C 180,E1 1273.093,E2 1273.093} C_VEL
LIN {X 0,Y 40.996,Z 1137.248,A -85,B 0,C 180,E1 1259.737,E2 1259.737} C_VEL
LIN {X 0,Y 46.018,Z 1136.646,A -85,B 0,C 180,E1 1258.199,E2 1258.199} C_VEL
LIN {X 0,Y 34.47,Z 1137.921,A -85,B 0,C 180,E1 1253.948,E2 1253.948} C_VEL
LIN {X 0,Y 27.175,Z 1138.617,A -85,B 0,C 180,E1 1251.702,E2 1251.702} C_VEL
LIN {X 0,Y 13.253,Z 1139.435,A -85,B 0,C 180,E1 1253.516,E2 1253.516} C_VEL
LIN {X 0,Y 3.035,Z 1139.709,A -85,B 0,C 180,E1 1258.692,E2 1258.692} C_VEL
LIN {X 0,Y 0.355,Z 1139.762,A -85,B 0,C 180,E1 1246.929,E2 1246.929} C_VEL
LIN {X 0,Y 0.727,Z 1139.763,A -85,B 0,C 180,E1 1084.93,E2 1084.93} C_VEL
LIN {X 0,Y 0.727,Z 1139.755,A -85,B 0,C 180,E1 1255.07,E2 1255.07} C_VEL
LIN {X 0,Y 0.355,Z 1139.762,A -85,B 0,C 180,E1 1246.929,E2 1246.929} C_VEL
LIN {X 0,Y 1.624,Z 1141.762,A -85,B 0,C 180,E1 1086.119,E2 1086.119} C_VEL
LIN {X 0,Y 1.624,Z 1164.5,A -85,B 0,C 180,E1 1086.119,E2 1086.119} C_VEL
LIN {X 0,Y 1.624,Z 1164.5,A -85,B 0,C 180,E1 1086.119,E2 1086.119}

QRS_NEXT_CUT()

QRS_NEXT()
QRS_HOME()

END
